// TIA Portal V17 export
// export: Created 2023-04-04T07:17:24.4121272Z, ExportSetting WithDefaults, DisplayName Totally Integrated Automation Portal, DisplayVersion V17 Update 4, DisplayName TIA Portal Openness, DisplayVersion V17 Update 4, DisplayName TIA Portal Version Control Interface, DisplayVersion V17, DisplayName STEP 7 Professional, DisplayVersion V17 Update 4, DisplayName STEP 7 Safety, DisplayVersion V17, DisplayName WinCC Professional, DisplayVersion V17 Update 4
FUNCTION "SS Warnings" : Void   // FC103, LAD
{ S7_Optimized_Access := 'TRUE' }
VERSION : 0.1
// stored: AutoNumber false, IsIECCheckEnabled false, SetENOAutomatically false, UDAEnableTagReadback false
BEGIN

REGION Network 1: Warning Status On/Off
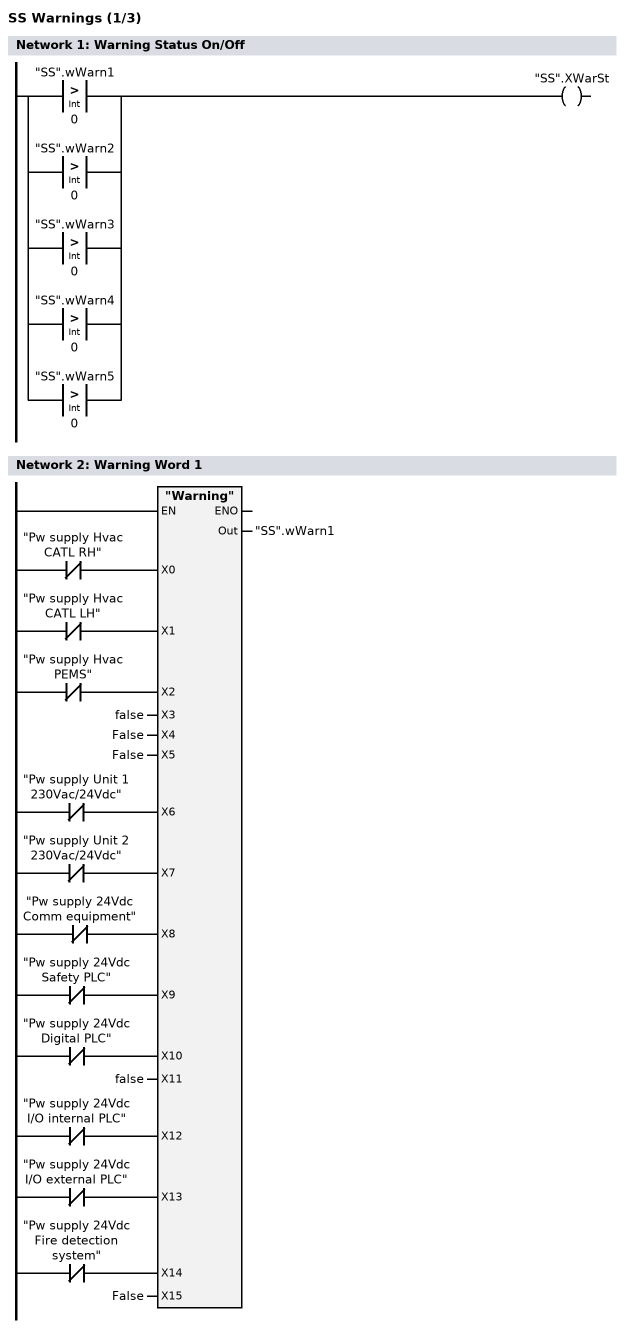
   RUNG wire#powerrail
      { S7_Templates := "SrcType := Int" } GT_Contact(in1 := "SS".wWarn1, in2 := 0)
      wire#w1
      Coil( "SS".XWarSt )
   END_RUNG
   RUNG wire#powerrail
      { S7_Templates := "SrcType := Int" } GT_Contact(in1 := "SS".wWarn2, in2 := 0)
   END_RUNG wire#w1
   RUNG wire#powerrail
      { S7_Templates := "SrcType := Int" } GT_Contact(in1 := "SS".wWarn3, in2 := 0)
   END_RUNG wire#w1
   RUNG wire#powerrail
      { S7_Templates := "SrcType := Int" } GT_Contact(in1 := "SS".wWarn4, in2 := 0)
   END_RUNG wire#w1
   RUNG wire#powerrail
      { S7_Templates := "SrcType := Int" } GT_Contact(in1 := "SS".wWarn5, in2 := 0)
   END_RUNG wire#w1
   // the same network as SCL:
   "SS".XWarSt := ("SS".wWarn1 > 0) OR ("SS".wWarn2 > 0) OR ("SS".wWarn3 > 0) OR ("SS".wWarn4 > 0) OR ("SS".wWarn5 > 0);
END_REGION

REGION Network 2: Warning Word 1
   RUNG wire#powerrail
      "Warning"(X0 := wire#w1, X1 := wire#w2, X2 := wire#w3, X6 := wire#w4, X7 := wire#w5, X8 := wire#w6, X9 := wire#w7, X10 := wire#w8, X12 := wire#w9, X13 := wire#w10, X14 := wire#w11, X3 := false, X4 := False, X5 := False, X11 := false, X15 := False, Out => "SS".wWarn1)
   END_RUNG
   RUNG wire#powerrail
      I_Contact( "Pw supply Hvac CATL RH" )
   END_RUNG wire#w1
   RUNG wire#powerrail
      I_Contact( "Pw supply Hvac CATL LH" )
   END_RUNG wire#w2
   RUNG wire#powerrail
      I_Contact( "Pw supply Hvac PEMS" )
   END_RUNG wire#w3
   RUNG wire#powerrail
      I_Contact( "Pw supply Unit 1 230Vac/24Vdc" )
   END_RUNG wire#w4
   RUNG wire#powerrail
      I_Contact( "Pw supply Unit 2 230Vac/24Vdc" )
   END_RUNG wire#w5
   RUNG wire#powerrail
      I_Contact( "Pw supply 24Vdc Comm equipment" )
   END_RUNG wire#w6
   RUNG wire#powerrail
      I_Contact( "Pw supply 24Vdc Safety PLC" )
   END_RUNG wire#w7
   RUNG wire#powerrail
      I_Contact( "Pw supply 24Vdc Digital PLC" )
   END_RUNG wire#w8
   RUNG wire#powerrail
      I_Contact( "Pw supply 24Vdc I/O internal PLC" )
   END_RUNG wire#w9
   RUNG wire#powerrail
      I_Contact( "Pw supply 24Vdc I/O external PLC" )
   END_RUNG wire#w10
   RUNG wire#powerrail
      I_Contact( "Pw supply 24Vdc Fire detection system" )
   END_RUNG wire#w11
   // the same network as SCL:
   "Warning"(X0 := NOT "Pw supply Hvac CATL RH",
             X1 := NOT "Pw supply Hvac CATL LH",
             X2 := NOT "Pw supply Hvac PEMS",
             X3 := false,
             X4 := False,
             X5 := False,
             X6 := NOT "Pw supply Unit 1 230Vac/24Vdc",
             X7 := NOT "Pw supply Unit 2 230Vac/24Vdc",
             X8 := NOT "Pw supply 24Vdc Comm equipment",
             X9 := NOT "Pw supply 24Vdc Safety PLC",
             X10 := NOT "Pw supply 24Vdc Digital PLC",
             X11 := false,
             X12 := NOT "Pw supply 24Vdc I/O internal PLC",
             X13 := NOT "Pw supply 24Vdc I/O external PLC",
             X14 := NOT "Pw supply 24Vdc Fire detection system",
             X15 := False,
             Out => "SS".wWarn1);
END_REGION

REGION Network 3: Warning Word 2
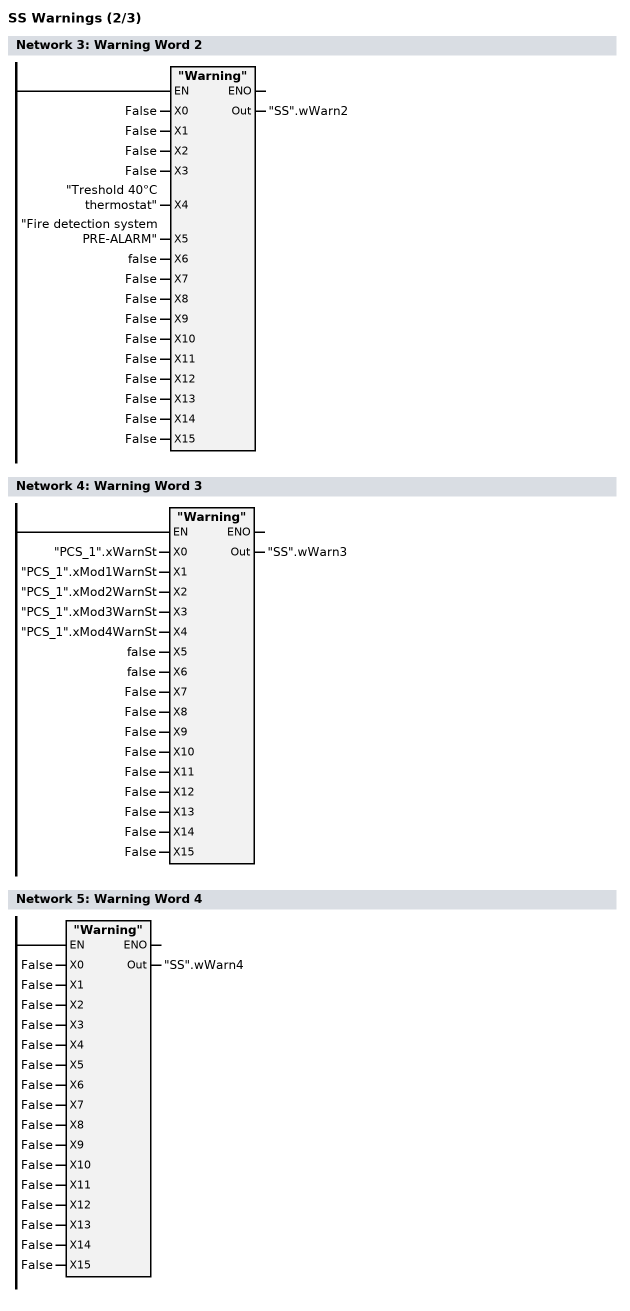
   RUNG wire#powerrail
      "Warning"(X0 := False, X1 := False, X2 := False, X3 := False, X4 := "Treshold 40°C thermostat", X5 := "Fire detection system PRE-ALARM", X6 := false, X7 := False, X8 := False, X9 := False, X10 := False, X11 := False, X12 := False, X13 := False, X14 := False, X15 := False, Out => "SS".wWarn2)
   END_RUNG
   // the same network as SCL:
   "Warning"(X0 := False,
             X1 := False,
             X2 := False,
             X3 := False,
             X4 := "Treshold 40°C thermostat",
             X5 := "Fire detection system PRE-ALARM",
             X6 := false,
             X7 := False,
             X8 := False,
             X9 := False,
             X10 := False,
             X11 := False,
             X12 := False,
             X13 := False,
             X14 := False,
             X15 := False,
             Out => "SS".wWarn2);
END_REGION

REGION Network 4: Warning Word 3
   RUNG wire#powerrail
      "Warning"(X0 := "PCS_1".xWarnSt, X1 := "PCS_1".xMod1WarnSt, X2 := "PCS_1".xMod2WarnSt, X3 := "PCS_1".xMod3WarnSt, X4 := "PCS_1".xMod4WarnSt, X5 := false, X6 := false, X7 := False, X8 := False, X9 := False, X10 := False, X11 := False, X12 := False, X13 := False, X14 := False, X15 := False, Out => "SS".wWarn3)
   END_RUNG
   // the same network as SCL:
   "Warning"(X0 := "PCS_1".xWarnSt,
             X1 := "PCS_1".xMod1WarnSt,
             X2 := "PCS_1".xMod2WarnSt,
             X3 := "PCS_1".xMod3WarnSt,
             X4 := "PCS_1".xMod4WarnSt,
             X5 := false,
             X6 := false,
             X7 := False,
             X8 := False,
             X9 := False,
             X10 := False,
             X11 := False,
             X12 := False,
             X13 := False,
             X14 := False,
             X15 := False,
             Out => "SS".wWarn3);
END_REGION

REGION Network 5: Warning Word 4
   RUNG wire#powerrail
      "Warning"(X0 := False, X1 := False, X2 := False, X3 := False, X4 := False, X5 := False, X6 := False, X7 := False, X8 := False, X9 := False, X10 := False, X11 := False, X12 := False, X13 := False, X14 := False, X15 := False, Out => "SS".wWarn4)
   END_RUNG
   // the same network as SCL:
   "Warning"(X0 := False,
             X1 := False,
             X2 := False,
             X3 := False,
             X4 := False,
             X5 := False,
             X6 := False,
             X7 := False,
             X8 := False,
             X9 := False,
             X10 := False,
             X11 := False,
             X12 := False,
             X13 := False,
             X14 := False,
             X15 := False,
             Out => "SS".wWarn4);
END_REGION

REGION Network 6: Warning Word 5
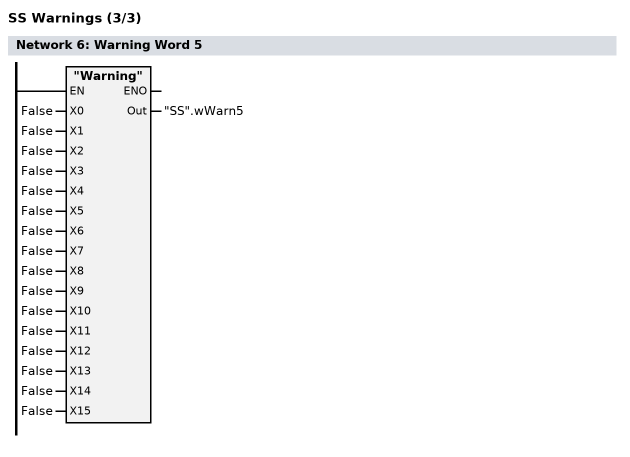
   RUNG wire#powerrail
      "Warning"(X0 := False, X1 := False, X2 := False, X3 := False, X4 := False, X5 := False, X6 := False, X7 := False, X8 := False, X9 := False, X10 := False, X11 := False, X12 := False, X13 := False, X14 := False, X15 := False, Out => "SS".wWarn5)
   END_RUNG
   // the same network as SCL:
   "Warning"(X0 := False,
             X1 := False,
             X2 := False,
             X3 := False,
             X4 := False,
             X5 := False,
             X6 := False,
             X7 := False,
             X8 := False,
             X9 := False,
             X10 := False,
             X11 := False,
             X12 := False,
             X13 := False,
             X14 := False,
             X15 := False,
             Out => "SS".wWarn5);
END_REGION
END_FUNCTION
